{attribute 'linkalways'}
{attribute 'no_explicit_call' := 'This FB is a CLASS and must be accessed using methods or properties'}
{attribute 'enable_dynamic_creation'}
FUNCTION_BLOCK _ETcVnEdgeSelection EXTENDS EnumDatatypeBase
VAR
	localData : ETcVnEdgeSelection;
	activeData : REFERENCE TO ETcVnEdgeSelection;
	enumBaseDatatype : _DINT(localData);
END_VAR

METHOD PRIVATE AddLocalEnumeration
VAR_INPUT
	Enumeration : T_MAXSTRING;
	Value : ETcVnEdgeSelection;
END_VAR
AddEnumeration(Enumeration, Value);
END_METHOD

PROPERTY PUBLIC Address : PVOID
GET
Address := ADR(activeData);
END_GET
END_PROPERTY

METHOD PUBLIC ClearReference
VAR_INPUT
END_VAR
activeData REF= localData;
SetBaseDatatypeReference();
END_METHOD

METHOD PUBLIC Clone : I_Datatype
VAR
    pClone : POINTER TO _ETcVnEdgeSelection;
END_VAR
pClone := __NEW(_ETcVnEdgeSelection(InitialValue := Value));
IF pClone = 0 THEN
    RETURN;
END_IF
Clone := pClone^;
END_METHOD

METHOD FB_init : BOOL
VAR_INPUT
	bInitRetains : BOOL; // if TRUE, the retain variables are initialized (warm start / cold start)
	bInCopyCode : BOOL;  // if TRUE, the instance afterwards gets moved into the copy code (online change)
	InitialValue : ETcVnEdgeSelection;
END_VAR
localData := InitialValue;
AddBaseDatatype(enumBaseDatatype);
ClearReference();

AddLocalEnumeration('TCVN_ES_RISING', ETcVnEdgeSelection.TCVN_ES_RISING);
AddLocalEnumeration('TCVN_ES_FALLING', ETcVnEdgeSelection.TCVN_ES_FALLING);
AddLocalEnumeration('TCVN_ES_ANY', ETcVnEdgeSelection.TCVN_ES_ANY);
END_METHOD

PROPERTY PUBLIC Identifier : T_MAXSTRING
GET
Identifier := 'ETcVnEdgeSelection';
END_GET
END_PROPERTY

METHOD IsEnumeratorValueEqual : BOOL
VAR_INPUT
	Enumerator : I_KeyValueForwardEnumerator;
END_VAR
VAR
	storedValue : ETcVnEdgeSelection;
END_VAR
IF NOT Enumerator.TryGet(storedValue) THEN
	RETURN;
END_IF

IsEnumeratorValueEqual := storedValue = activeData;
END_METHOD

METHOD PUBLIC MakeReferenceTo
VAR_INPUT
	ReferenceTarget : REFERENCE TO ETcVnEdgeSelection;
END_VAR
activeData REF= ReferenceTarget;
SetBaseDatatypeReference();
END_METHOD

METHOD PROTECTED SetBaseDatatypeReference
VAR_INPUT
END_VAR
enumBaseDatatype.MakeReferenceTo(activeData);
END_METHOD

PROPERTY PUBLIC Size : UDINT
GET
Size := SIZEOF(activeData);
END_GET
END_PROPERTY

METHOD TryMakeReferenceTo : BOOL
VAR_INPUT
	Target : I_Datatype;
END_VAR
VAR
	pTargetData : POINTER TO ETcVnEdgeSelection;
END_VAR
IF NOT IsEquivalentTo(Target) THEN
	RETURN;
END_IF

pTargetData := Target.Address;
activeData REF= pTargetData^;
SetBaseDatatypeReference();
TryMakeReferenceTo := TRUE;
END_METHOD

PROPERTY PUBLIC Value : ETcVnEdgeSelection
GET
Value := activeData;
END_GET
SET
activeData := Value;
END_SET
END_PROPERTY

END_FUNCTION_BLOCK

(* stored: Version 1.1.0.1, ProductVersion 3.1.4026.13
   POU _ETcVnEdgeSelection: Id {adddb95e-990f-4b79-850e-03f705b821ed}, SpecialFunc None
   Folder Core: Id {786e59e2-ab1c-467b-b932-629f3a325cab}
   Folder Protected: Id {ad63e4e3-7aee-4ebb-9c62-9222358de0b5}
   Folder Customize: Id {e1794e2c-86d7-4b79-a8e7-3899ace27c68}
   Folder Constructor: Id {011bca42-c7e9-4a74-9bec-ee3316b73ddc}
   Folder Private: Id {48c68283-ded5-4197-9724-34c0036a153f}
   Folder Protected: Id {5a28fda5-d47c-4a1f-b1f1-642ce5a15823}
   Method AddLocalEnumeration: Id {57953eac-a450-46d8-85ef-4629e79f664a}
   Property Address: Id {304b2876-6538-4b51-a68a-141b07643039}
   Get Get: Id {58346331-e066-4252-be4b-0bb9de661313}
   Method ClearReference: Id {5cb76329-ff16-4da2-9bba-8bd96a51099c}
   Method Clone: Id {58c51f02-c159-425b-9bde-6aa508fd8def}
   Method FB_init: Id {8b13c906-288f-46b3-bf55-de442d777538}
   Property Identifier: Id {a61597f3-952a-4dbe-83fd-1c10a575262a}
   Get Get: Id {a2aebaba-813a-475a-8da2-2aba449b6689}
   Method IsEnumeratorValueEqual: Id {eef1a112-7164-40ab-a523-4cd23f691cd9}
   Method MakeReferenceTo: Id {6acf2196-1aaf-4a95-a9c1-7d192882f4cc}
   Method SetBaseDatatypeReference: Id {8d3f38d3-6a3c-48f1-a14b-bc56ac6cf5be}
   Property Size: Id {1adcbd0d-1772-425a-bb8b-c3c9e79cd410}
   Get Get: Id {bd5e0a88-a882-4437-a633-6449ce24ca72}
   Method TryMakeReferenceTo: Id {66cee595-6367-4009-900c-375aaed096f4}
   Property Value: Id {0912c759-6784-4fcb-be1c-aeec1720e0d1}
   Get Get: Id {ec401f1b-4064-49ef-97b2-46ae3eb5273d}
   Set Set: Id {f054d674-0296-4090-92f9-15279e642ed2} *)
